TYPE TAxisState :
	(	AS_PowerOff,
		AS_Powering,
		AS_NotHomed,
		AS_Homing,
		AS_InPosition,
		AS_Moving,
		AS_MovingHoming,
		AS_MovingLimitNeg,
		AS_OnLimitNeg,
		AS_Stopping,
		AS_InError,
		AS_Resetting
	);
END_TYPE

(* stored: Version 1.1.0.1, ProductVersion 3.1.4022.12
   DUT TAxisState: Id {b4066bd0-8b36-481f-81c3-d8886f82ec4c} *)
